(* IEC 61131-3 sources: CodesysTest/export/Function Blocks/FB_MachineCounter/FB_MachineCounter.pou, 3 files *)

(* ---- FB_MachineCounter.pou.st ---- *)
(*#-#-#-#-#-#-#-#-#-#---Declaration---#-#-#-#-#-#-#-#-#-#-#-#-#*)

FUNCTION_BLOCK FINAL FB_MachineCounter EXTENDS FB_BaseObject IMPLEMENTS ICounter
VAR_INPUT
END_VAR
VAR_OUTPUT
END_VAR
VAR PERSISTENT RETAIN
    count : UDINT;
END_VAR
(*#-#-#-#-#-#-#-#-#-#---Implementation---#-#-#-#-#-#-#-#-#-#-#-#-#*)

(* ---- AddToCount.m.st ---- *)
(*#-#-#-#-#-#-#-#-#-#---Declaration---#-#-#-#-#-#-#-#-#-#-#-#-#*)

METHOD AddToCount
VAR_INPUT
	amountToAdd : UDINT;
END_VAR
(*#-#-#-#-#-#-#-#-#-#---Implementation---#-#-#-#-#-#-#-#-#-#-#-#-#*)

count := count + amountToAdd;

(* ---- SetCount.m.st ---- *)
(*#-#-#-#-#-#-#-#-#-#---Declaration---#-#-#-#-#-#-#-#-#-#-#-#-#*)

METHOD SetCount
VAR_INPUT
	countSetting : UDINT;
END_VAR
(*#-#-#-#-#-#-#-#-#-#---Implementation---#-#-#-#-#-#-#-#-#-#-#-#-#*)

count := countSetting;
